Universal Robots PolyScope program: pop.urp

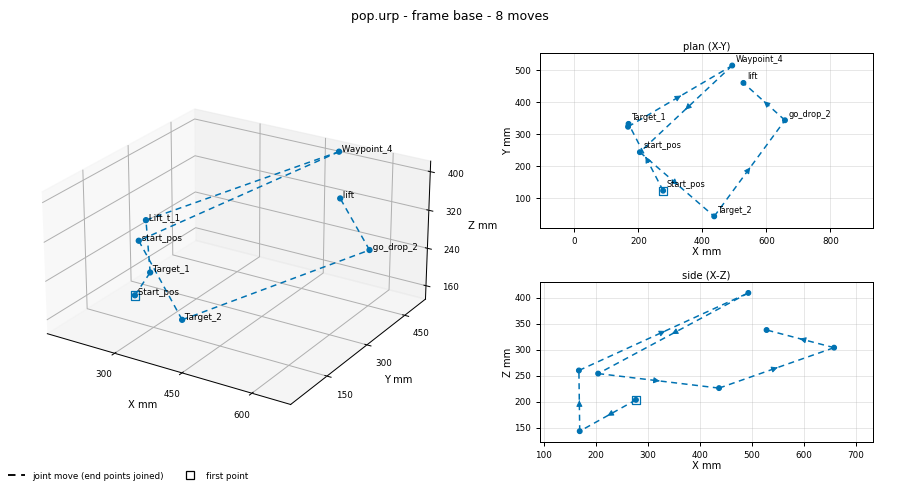
[picture p0: tool path of pop.urp in frame base, 8 of 8 moves have a stored position in this frame; points joined in program order, loops and branches not executed]
Program pop (installation=dev_test directory=/ursim/programs/scripts/manual createdIn=3.15.6.106324 lastSavedIn=3.15.8.106339 robotSerialNumber=2018359999)
Calibrated DH parameters: a=[0.000173, -0.08184, -0.390569, 0.000014, 0.000061, 0]; d=[0.089465, 325.63058, -320.968373, -4.551618, 0.094907, 0.082699]; alpha=[1.570634, -0.001282, 0.007518, 1.570171, -1.57068, 0]; deltaTheta=[0.000011, -1.377212, 1.46664, -0.089508, -0.000013, 0.000027]
Robot Program (runOnlyOnce=false)
  MoveJ speed 60 deg/s, acceleration 80 deg/s^2 (useActiveTCP=true)
    Script file /ursim/programs/scripts/tool_actions/execute_gripping_action.script
      | def execute_gripping_action():
      | 
      |     popup("Gripper action commencing", title = "Gripper action", blocking = True)
      | 
      |     voltage = get_standard_analog_in(0)
      |     target_pose = pose_add(get_actual_tcp_pose(), p[0, 0, 0.1, 0, 0, 0]) #50 mm up
      |     if (voltage > 1.5):
      |         sleep(1.0)
      |         set_standard_digital_out(0, True)   #close gripper
      |         movel(target_pose)
      | 
      | 
      |     else:
      |         popup("Voltage too low - Gripper not activated - STOPPING", title = "FAILURE", blocking = True)
      |     end
      | end
    Script file /ursim/programs/scripts/tool_actions/execute_drop_action.script
      | def execute_drop_action():
      |     set_standard_digital_out(0, False)
      | end
    Waypoint Start_pos: TCP in base x=277.303 y=122.945 z=203.701 mm, rx=3.0209 ry=-0.6146 rz=-0.0595 rad; joints [45, -70, -140, -64, 90.003, -22] deg
    Waypoint Target_1: TCP in base x=169.329 y=331.744 z=143.526 mm, rx=-3.0072 ry=-0.3161 rz=-0.051 rad; joints [80, -90, -140, -33, 90, -22] deg
    Script file /ursim/programs/scripts/tool_actions/grip_action.script
      | execute_gripping_action()
    Waypoint Lift_t_1: TCP in base x=167.741 y=322.739 z=260.168 mm, rx=-3.0319 ry=-0.3992 rz=-0.0402 rad; joints [80, -75, -130, -60, 90, -25] deg
    Waypoint Waypoint_4: TCP in base x=493.182 y=514.04 z=409.085 mm, rx=-3.06 ry=0.3486 rz=-0.0513 rad; joints [55, -120, -56, -90, 90, -22] deg
    Script file /ursim/programs/scripts/tool_actions/drop_action.script
      | execute_drop_action()
    Waypoint start_pos: TCP in base x=204.735 y=243.359 z=254.191 mm, rx=2.9436 ry=0.0514 rz=-0.1108 rad; joints [70, -70, -130, -82, 89.997, -22] deg
    Waypoint Target_2: TCP in base x=436.914 y=42.869 z=226.291 mm, rx=2.8016 ry=-1.2473 rz=-0.1156 rad; joints [20, -90, -120, -66, 90, -22] deg
    Script file /ursim/programs/scripts/tool_actions/grip_action.script
      | execute_gripping_action()
    Waypoint go_drop_2: TCP in base x=657.914 y=343.086 z=303.982 mm, rx=-2.9391 ry=0.8428 rz=-0.0987 rad; joints [36, -125, -64, -75, 90, -22] deg
    Script file /ursim/programs/scripts/tool_actions/drop_action.script
      | execute_drop_action()
    Waypoint lift: TCP in base x=528.213 y=459.693 z=337.901 mm, rx=3.0375 ry=-0.4811 rz=-0.0607 rad; joints [50, -120, -64.389, -90, 90, -22] deg
